// TIA Portal V20 export
VAR_GLOBAL   // PLC tag table "Lift"
   oLift_Actuators_Push AT %Q5100.0 : Bool;
   oLift_Actuator_Pull AT %Q5100.1 : Bool;
   iLift_SenA AT %I5100.0 : Bool;
   iLift_SenB AT %I5100.1 : Bool;
   iLift_SenC AT %I5100.2 : Bool;
   iLift_SenD AT %I5100.3 : Bool;
   iLift_Clamp1_Close AT %I5100.4 : Bool;
   iLift_Clamp1_Open AT %I5100.5 : Bool;
   iLift_Clamp2_Close AT %I5100.6 : Bool;
   iLift_Clamp2_Open AT %I5100.7 : Bool;
   iLift_Up_Position AT %I5101.0 : Bool;
   iLift_Down_Position AT %I5101.1 : Bool;
   iLift_Actuator1_Push AT %I5101.2 : Bool;
   iLift_Actuator1_Pull AT %I5101.3 : Bool;
   iLift_Actuator2_Push AT %I5101.4 : Bool;
   iLift_Actuator2_Pull AT %I5101.5 : Bool;
   iLift_Actuator3_Push AT %I5101.6 : Bool;
   iLift_Actuator3_Pull AT %I5101.7 : Bool;
   iLift_Actuator4_Push AT %I5102.0 : Bool;
   iLift_Actuator4_Pull AT %I5102.1 : Bool;
   QR_ReaderST34 AT %ID5002 : DInt;
   QR_ReaderST32 AT %ID5012 : DInt;
END_VAR
